{attribute 'qualified_only'}
{attribute 'strict'}
TYPE E_StatesTop :
(
	Disabled	:=	10000,
	Enabled		:=	20000
) DINT;
END_TYPE

(* stored: Version 1.1.0.1, ProductVersion 3.1.4022.18
   DUT E_StatesTop: Id {5369fa98-da0c-4000-a711-9460e8401e23} *)
